// TwinCAT 3 PLC project EnOcean_Sample_CX9020
// libraries:
//   Tc2_EnOcean, * (Beckhoff Automation GmbH)
//   Tc2_Standard, * (Beckhoff Automation GmbH)
//   Tc2_System, * (Beckhoff Automation GmbH)
//   Tc3_Module, * (Beckhoff Automation GmbH)
// project tree:
//   Global Variables/ Globale_Variablen.TcGVL, Variablen_Konfiguration.TcGVL
//   POUs/ MAIN.TcPOU (not stored)
//   / Standard.TcTTO (not stored)

// ---- Global Variables/Globale_Variablen.TcGVL
{attribute 'Tc2GvlVarNames'}
VAR_GLOBAL
	st6581Input  AT %I* : KL6581_Input;
	st6581Output AT %Q* : KL6581_Output;
	stKL6581            : STR_KL6581;
END_VAR

// ---- Global Variables/Variablen_Konfiguration.TcGVL
{attribute 'Tc2GvlVarNames'}
VAR_CONFIG
END_VAR
